{attribute 'linkalways'} 
{attribute 'no_explicit_call' := 'This FB is a CLASS and must be accessed using methods or properties'}
{attribute 'enable_dynamic_creation'}
FUNCTION_BLOCK Node_F_VN_CompensateLensDistortionExp1 EXTENDS VisionNode
VAR
    ipSrcImage : _ITcVnImage;
    ipDestImage : _ITcVnImage;
    aCameraMatrix : _TcVnMatrix3x3_LREAL;
    aDistortionCoefficients : _TcVnArray8_LREAL;
    hrPrev : _HRESULT(S_OK);
	hresult : _HRESULT(S_OK);
END_VAR

METHOD PUBLIC  Clone : I_Node
VAR
	pNode : POINTER TO Node_F_VN_CompensateLensDistortionExp1;
END_VAR
pNode := __NEW(Node_F_VN_CompensateLensDistortionExp1);
Clone := pNode^;
END_METHOD

METHOD FB_init : BOOL
VAR_INPUT
	bInitRetains : BOOL; // if TRUE, the retain variables are initialized (warm start / cold start)
	bInCopyCode : BOOL;  // if TRUE, the instance afterwards gets moved into the copy code (online change)
END_VAR
AddInput('ipSrcImage', ipSrcImage);
AddInput('aCameraMatrix', aCameraMatrix);
AddInput('aDistortionCoefficients', aDistortionCoefficients);
AddInput('hrPrev', hrPrev);
AddOutput('ipDestImage', ipDestImage);
AddOutput('hresult', hresult);
END_METHOD

METHOD PROTECTED OnExecute
hresult.Value := F_VN_CompensateLensDistortionExp1(
    ipSrcImage := ipSrcImage.Value,
	ipDestImage := ipDestImage.Value,
    aCameraMatrix := aCameraMatrix.Value,
    aDistortionCoefficients := aDistortionCoefficients.Value,
	hrPrev := hrPrev.Value);
END_METHOD

METHOD PUBLIC PreExecutionCheck
VAR_INPUT
	Check : I_PreExecutionChecks;
END_VAR
Check.IsTrue(ipSrcImage.IsValid, 'ipSrcImage must contain an image');
END_METHOD

END_FUNCTION_BLOCK

(* stored: Version 1.1.0.1, ProductVersion 3.1.4024.15
   POU Node_F_VN_CompensateLensDistortionExp1: Id {e3a8051b-8851-0073-3775-37d2ca4dbb0d}, SpecialFunc None
   Folder Constructor: Id {573f2f31-f72f-0692-2b39-8dd636415df8}
   Method Clone: Id {ed10214a-327e-09e9-18bd-c339db4a7b96}
   Method FB_init: Id {a0df9156-eccb-0d47-1c47-2c90a3b8dd61}
   Method OnExecute: Id {316d58f2-e33d-04e0-1f73-9a7bf628402d}
   Method PreExecutionCheck: Id {f77b988a-c45d-0da3-1b63-c5388b2347b9} *)
